FUNCTION_BLOCK FB_HE_SATT_CommandsEpics IMPLEMENTS I_HE_SATT_Commands
VAR
    bPermitMove : BOOL;
    bReset : BOOL;
END_VAR


PROPERTY PermitMove : BOOL
GET

PermitMove := THIS^.bPermitMove;
END_GET
SET

THIS^.bPermitMove := PermitMove;
END_SET
END_PROPERTY


PROPERTY Reset : BOOL
GET

Reset := THIS^.bReset;
END_GET
SET

THIS^.bReset := Reset;
END_SET
END_PROPERTY

END_FUNCTION_BLOCK

(* stored: Version 1.1.0.1
   POU FB_HE_SATT_CommandsEpics: Id {438d1cad-cb94-4f9e-b53f-7bd18ce892e3}, SpecialFunc None
   Property PermitMove: Id {bde7f3ef-5c59-462a-8b06-ebaa73a456bb}
   Get Get: Id {b8a740ce-11c5-4a17-bf5b-7fbe705aeb0e}
   Set Set: Id {a57ce744-269a-4c7f-98cb-fb53586ebfc3}
   Property Reset: Id {f99b62d3-c285-4fb4-bcb3-07b82fb8641c}
   Get Get: Id {7eae352d-6f12-4763-b39d-cc3c03ad0c23}
   Set Set: Id {c638c8b8-8043-40d4-ad97-ab3bb05aa75e} *)
